(* IEC 61131-3 sources: Stat_Resistant_AI_Coding/src/plc/common, 4 files *)

(* ---- FB_MainPressureControl.st ---- *)
(*
  Canonical AI-owned POU source.
  Deploy only through PLC Engineering MCP and verify by readback + compile.
*)

(* ===== DECLARATION ===== *)
FUNCTION_BLOCK FB_MainPressureControl
VAR_INPUT
  /// Enable monitoring only after Station is OPERATIONAL and the I/O bus is OK
  xMonitoringEnabled : BOOL;
  /// Electrical safety circuit feedback from ControlOn.OutImm.IsCtrlOn
  xControlOnOk       : BOOL;
  /// Additional application interlock for opening the master air valve
  xValveRelease      : BOOL;
  /// Pressure below the lower threshold (primary MAX < 0.3 bar)
  xPressureLow       : BOOL;
  /// Pressure above the upper threshold (primary MAX > 4.5 bar)
  xPressureHigh      : BOOL;
  /// Maximum time allowed for each pressure transition
  tMonitoringTime   : TIME := T#5S;
END_VAR
VAR_OUTPUT
  /// Command for the master air valve _000K085A
  xValveOn                : BOOL;
  /// TRUE when the valve is on and only the high-pressure feedback is active
  xPressureReady          : BOOL;
  /// Connect to ControlOn.ParImm.UserEnableControlOn
  xEnableControlOn        : BOOL;
  /// Latched fault: pressure did not reach the upper threshold
  xFaultPressureNotHigher : BOOL;
  /// Latched fault: pressure did not reach the lower threshold
  xFaultPressureNotLower  : BOOL;
  /// Current plausibility error: both pressure switches are active
  xPressureSignalConflict : BOOL;
END_VAR
VAR
  _timerPressureHigh : TON;
  _timerPressureLow  : TON;
END_VAR

(* ===== IMPLEMENTATION ===== *)
// Outside the valid application/I/O state, actively close the valve and do not
// evaluate uninitialized bus inputs.
IF ( NOT xMonitoringEnabled )
THEN
  _timerPressureHigh(IN := FALSE, PT := tMonitoringTime);
  _timerPressureLow(IN := FALSE, PT := tMonitoringTime);

  xValveOn                := FALSE;
  xPressureReady          := FALSE;
  xEnableControlOn        := FALSE;
  xFaultPressureNotHigher := FALSE;
  xFaultPressureNotLower  := FALSE;
  xPressureSignalConflict := FALSE;
  RETURN;
END_IF

// The two pressure switches describe mutually exclusive pressure ranges.
xPressureSignalConflict := ( xPressureLow ) AND
                           ( xPressureHigh );

// Monitor the feedback that belongs to the actual valve command.
// During a normal transition both feedback signals may temporarily be FALSE.
_timerPressureHigh(
  IN := ( xValveOn ) AND
        ( NOT ( ( xPressureHigh ) AND ( NOT xPressureLow ) ) ),
  PT := tMonitoringTime
);

_timerPressureLow(
  IN := ( NOT xValveOn ) AND
        ( NOT ( ( xPressureLow ) AND ( NOT xPressureHigh ) ) ),
  PT := tMonitoringTime
);

// A contradictory feedback is diagnosed immediately. Transition faults use
// the configured delay. Faults remain latched until Control On is removed and
// a plausible depressurized state has been reached.
IF ( xPressureSignalConflict )
THEN
  xFaultPressureNotHigher := TRUE;
  xFaultPressureNotLower  := TRUE;
ELSE
  IF ( _timerPressureHigh.Q )
  THEN
    xFaultPressureNotHigher := TRUE;
  END_IF

  IF ( _timerPressureLow.Q )
  THEN
    xFaultPressureNotLower := TRUE;
  END_IF
END_IF

IF ( NOT xControlOnOk ) AND
   ( xPressureLow ) AND
   ( NOT xPressureHigh )
THEN
  xFaultPressureNotHigher := FALSE;
  xFaultPressureNotLower  := FALSE;
END_IF

// Fail-safe output behavior:
// - no electrical Control On feedback => close the valve
// - missing application release => close the valve
// - any pressure fault => close the valve
// - opening is permitted only from a plausible depressurized state
IF ( NOT xControlOnOk ) OR
   ( NOT xValveRelease ) OR
   ( xFaultPressureNotHigher ) OR
   ( xFaultPressureNotLower )
THEN
  xValveOn := FALSE;
ELSIF ( NOT xValveOn ) AND
      ( xPressureLow ) AND
      ( NOT xPressureHigh )
THEN
  xValveOn := TRUE;
END_IF

xPressureReady := ( xValveOn ) AND
                  ( xValveRelease ) AND
                  ( xPressureHigh ) AND
                  ( NOT xPressureLow ) AND
                  ( NOT xFaultPressureNotHigher ) AND
                  ( NOT xFaultPressureNotLower );

xEnableControlOn := ( NOT xFaultPressureNotHigher ) AND
                    ( NOT xFaultPressureNotLower );

(* ---- FB_MaintenanceDoorControl.st ---- *)
(*
  Canonical AI-owned POU source.
  Deploy only through PLC Engineering MCP and verify by readback + compile.
*)

(* ===== DECLARATION ===== *)
FUNCTION_BLOCK FB_MaintenanceDoorControl
VAR_INPUT
  /// Cyclic execution enable; normally Station OPERATIONAL and fieldbus OK
  xEnable             : BOOL;
  /// Raw Control On push-button request
  xControlOnRequest   : BOOL;
  /// Confirmed electrical Control On state; keeps both locks energized
  xControlOnOk        : BOOL;
  /// Feedback: maintenance door A is closed
  xDoorAClosed        : BOOL;
  /// Feedback: maintenance door B is closed
  xDoorBClosed        : BOOL;
  /// Feedback: maintenance-door safety relay is energized
  xMaintenanceRelayFeedback : BOOL;
  /// Maximum time for both lock feedbacks to become active
  tLockMonitoringTime : TIME := T#5S;
  /// Maximum delay from both doors closed to safety-relay feedback
  tRelayMonitoringTime : TIME := T#1S;
END_VAR
VAR_OUTPUT
  /// Command for maintenance door A lock
  xDoorLockAOn          : BOOL;
  /// Command for maintenance door B lock
  xDoorLockBOn          : BOOL;
  /// TRUE only when both maintenance-door closed feedbacks are active
  xAllDoorsClosed       : BOOL;
  /// Additional release for the main-pressure valve
  xMainPressureRelease  : BOOL;
  /// Latched aggregate maintenance-door interlock fault
  xFaultDoorNotLocked   : BOOL;
  /// Latched detail: maintenance door A closed feedback was missing
  xFaultDoorANotClosed  : BOOL;
  /// Latched detail: maintenance door B closed feedback was missing
  xFaultDoorBNotClosed  : BOOL;
  /// Latched detail: safety-relay feedback was missing after both doors closed
  xFaultRelayFeedbackMissing : BOOL;
END_VAR
VAR
  _timerDoorLock      : TON;
  _timerRelayFeedback : TON;
END_VAR

(* ===== IMPLEMENTATION ===== *)
// This FB contains no project BMKs. The caller connects the two lock
// outputs, two feedbacks and the standard ControlOn signals.
IF ( NOT xEnable )
THEN
  _timerDoorLock(IN := FALSE, PT := tLockMonitoringTime);
  _timerRelayFeedback(IN := FALSE, PT := tRelayMonitoringTime);

  xDoorLockAOn         := FALSE;
  xDoorLockBOn         := FALSE;
  xAllDoorsClosed      := FALSE;
  xMainPressureRelease := FALSE;
  xFaultDoorNotLocked  := FALSE;
  xFaultDoorANotClosed := FALSE;
  xFaultDoorBNotClosed := FALSE;
  xFaultRelayFeedbackMissing := FALSE;
  RETURN;
END_IF

// Energize both locks while the operator presses Control On. Once the
// electrical Control On feedback is present, keep the locks energized after
// the momentary push-button is released.
xDoorLockAOn := ( xControlOnRequest ) OR
                ( xControlOnOk );
xDoorLockBOn := ( xControlOnRequest ) OR
                ( xControlOnOk );

xAllDoorsClosed := ( xDoorAClosed ) AND
                   ( xDoorBClosed );

// Start one shared monitoring time as soon as both lock outputs are requested.
// A loss of either feedback while Control On remains active starts the same
// monitoring again.
_timerDoorLock(
  IN := ( xDoorLockAOn ) AND
        ( xDoorLockBOn ) AND
        ( NOT xAllDoorsClosed ),
  PT := tLockMonitoringTime
);

IF ( _timerDoorLock.Q )
THEN
  IF ( NOT xDoorAClosed )
  THEN
    xFaultDoorANotClosed := TRUE;
  END_IF

  IF ( NOT xDoorBClosed )
  THEN
    xFaultDoorBNotClosed := TRUE;
  END_IF
END_IF

// Once both door-closed inputs are present, the maintenance safety relay must
// confirm the electrical safety circuit within one second.
_timerRelayFeedback(
  IN := ( xDoorLockAOn ) AND
        ( xDoorLockBOn ) AND
        ( xAllDoorsClosed ) AND
        ( NOT xMaintenanceRelayFeedback ),
  PT := tRelayMonitoringTime
);

IF ( _timerRelayFeedback.Q )
THEN
  xFaultRelayFeedbackMissing := TRUE;
END_IF

// Keep the fault latched until the lock request has been removed. This gives
// the Station event the same deliberate Control Off/reset lifecycle as the
// main-pressure faults.
IF ( NOT xDoorLockAOn ) AND
   ( NOT xDoorLockBOn )
THEN
  xFaultDoorANotClosed          := FALSE;
  xFaultDoorBNotClosed          := FALSE;
  xFaultRelayFeedbackMissing    := FALSE;
END_IF

xFaultDoorNotLocked := ( xFaultDoorANotClosed ) OR
                       ( xFaultDoorBNotClosed ) OR
                       ( xFaultRelayFeedbackMissing );

// Pressure is released only when both commanded locks and both independent
// closed feedbacks are present. A latched timeout requires Control Off before
// a new pressure-on attempt.
xMainPressureRelease := ( xDoorLockAOn ) AND
                        ( xDoorLockBOn ) AND
                        ( xAllDoorsClosed ) AND
                        ( xMaintenanceRelayFeedback ) AND
                        ( NOT xFaultDoorNotLocked );

(* ---- FB_OperatorButton.st ---- *)
(*
  Canonical AI-owned POU source.
  Deploy only through PLC Engineering MCP and verify by readback + compile.
*)

(* ===== DECLARATION ===== *)
FUNCTION_BLOCK FB_OperatorButton
VAR_INPUT
  /// TRUE while the SFC step is requesting an operator acknowledgement
  Execute       : BOOL;
  /// Physical push-button signal
  ButtonPressed : BOOL;
  /// Shared 500 ms flash pulse, for example Station.FlashBits.Pulse500ms
  Blink500ms    : BOOL;
END_VAR
VAR_OUTPUT
  /// Latched completion; remains TRUE until Execute becomes FALSE
  Done          : BOOL;
  /// Command for the illuminated push-button lamp
  LampOn        : BOOL;
END_VAR

(* ===== IMPLEMENTATION ===== *)
// Execute follows the same lifecycle used by OpCon commands:
// FALSE ends the request and restores the initial state.
IF ( NOT Execute )
THEN
  Done   := FALSE;
  LampOn := FALSE;
  RETURN;
END_IF

// While waiting, flash the lamp. A detected button signal completes the
// request and switches the lamp off in the same PLC cycle.
IF ( NOT Done )
THEN
  IF ( ButtonPressed )
  THEN
    Done   := TRUE;
    LampOn := FALSE;
  ELSE
    LampOn := Blink500ms;
  END_IF
ELSE
  LampOn := FALSE;
END_IF

(* ---- FB_PressureFeedbackSimulation.st ---- *)
(*
  Canonical AI-owned POU source.
  Deploy only through PLC Engineering MCP and verify by readback + compile.
*)

(* ===== DECLARATION ===== *)
FUNCTION_BLOCK FB_PressureFeedbackSimulation
VAR_INPUT
  /// Enable the virtual feedback only while the Station and I/O bus are valid
  xEnable        : BOOL;
  /// Sustained electrical state from ControlOn.OutImm.IsCtrlOn
  xControlOn     : BOOL;
  /// Delay before changing to the pressure state requested by Control On/Off
  tSwitchDelay   : TIME := T#1S;
END_VAR
VAR_OUTPUT
  /// Virtual replacement for the unwired low-pressure switch
  xPressureLow      : BOOL;
  /// Virtual replacement for the unwired high-pressure switch
  xPressureHigh     : BOOL;
  /// TRUE while the one-second virtual pressure transition is running
  xTransitionActive : BOOL;
END_VAR
VAR
  _timerToHigh : TON;
  _timerToLow  : TON;
  _initialized : BOOL;
END_VAR

(* ===== IMPLEMENTATION ===== *)
// The physical pressure inputs are intentionally unwired. Disable both
// virtual inputs outside the valid application/I/O state and re-synchronize
// to the current ControlOn state when monitoring becomes valid again.
IF ( NOT xEnable )
THEN
  _timerToHigh(IN := FALSE, PT := tSwitchDelay);
  _timerToLow(IN := FALSE, PT := tSwitchDelay);

  xPressureLow      := FALSE;
  xPressureHigh     := FALSE;
  xTransitionActive := FALSE;
  _initialized      := FALSE;
  RETURN;
END_IF

// Initialization is not a Control On/Off transition. Adopt the current safe
// state immediately so Control On cannot occur before a virtual LOW exists.
IF ( NOT _initialized )
THEN
  xPressureLow  := ( NOT xControlOn );
  xPressureHigh := ( xControlOn );
  _initialized  := TRUE;
END_IF

// Keep the previous stable state during the delay, then switch LOW/HIGH in
// one PLC cycle. The outputs can therefore never both be TRUE.
_timerToHigh(
  IN := ( xControlOn ) AND
        ( NOT xPressureHigh ),
  PT := tSwitchDelay
);

_timerToLow(
  IN := ( NOT xControlOn ) AND
        ( NOT xPressureLow ),
  PT := tSwitchDelay
);

IF ( _timerToHigh.Q )
THEN
  xPressureHigh := TRUE;
  xPressureLow  := FALSE;
ELSIF ( _timerToLow.Q )
THEN
  xPressureLow  := TRUE;
  xPressureHigh := FALSE;
END_IF

xTransitionActive := ( ( xControlOn ) AND ( NOT xPressureHigh ) ) OR
                     ( ( NOT xControlOn ) AND ( NOT xPressureLow ) );
